TYPE ST_fbDiagnostics :
STRUCT
	asResults	:	ARRAY [1..20] OF STRING;
	resultIdx	:	FB_Index(
		InitVal := 1,
		UpperLImit := 20
	);
END_STRUCT
END_TYPE

(* stored: Version 1.1.0.1, ProductVersion 3.1.4018.5
   DUT ST_fbDiagnostics: Id {07dcfd66-d6ab-4320-bb04-7a16ac42f205} *)
